Fanuc KAREL source: compact_preamble.KL

PROGRAM KD00041
%NOLOCKGROUP
%ENVIRONMENT TPE
VAR
I:INTEGER;J:INTEGER;B:BOOLEAN;R:REAL;S : STRING[80]
-- UNRESOLVED DECLARATIONS (source type spelling not recovered)
-- D : TYPE_0x1100 (type_u16=0x1100)
BEGIN
I=1
END KD00041
